(* IEC 61131-3 sources: jiepp/tests/jiepp/input/counter_macro, 2 files *)

(* ---- a.iec ---- *)
{#include	"b.iec"}

program a{### __COUNTER__}
__COUNTER__;
end_program

(* ---- b.iec ---- *)
program b{### __COUNTER__}
__COUNTER__;
end_program
